SUBAPPLICATION Uebung_HystereseHorizontal_AX_withAnalog (* MID/DEAD/HYSTERESIS-Eingabefelder bewegen live die 5 Schwellwert-Dreiecke im horizontalen Bargraph (wie Uebung_225_AX fuer Workspace_Dreieck, aber 5 Marker statt 1 und mit AR-Arithmetik fuer die 4 abgeleiteten Schwellen) *)
  (* Standard: 61499-2; Description: Copyright (c) 2026 Meisterschulen am Ostbahnhof This program and the accompanying materials are made available under the terms of the Eclipse Public License 2.0 which is available at https://www.eclipse.org/legal/epl-2.0/ SPDX-License-Identifier: EPL-2.0 *)
  (* Version 1.0, 2026-09-26, Franz Höpfinger, Meisterschulen am Ostbahnhof, Franz: 3 Eingabefelder MID/DEAD/HYSTERESIS bewegen die 5 Schwellwert-Dreiecke live - Vorbild Uebung_225_AX (Dreieck-Sollwertmarker): NumericValue_PHYSA -> AR-Arithmetik -> AR_TO_AI -> Q_ChildPosition_AI. *)
  PACKAGE Uebungen;
  IMPORT Uebungen::const::UT::HystereseHorizontal::DefaultPool_Numeric::InputNumber_MID_N;
  IMPORT Uebungen::const::UT::HystereseHorizontal::DefaultPool_Numeric::InputNumber_DEAD_N;
  IMPORT Uebungen::const::UT::HystereseHorizontal::DefaultPool_Numeric::InputNumber_HYSTERESIS_N;
  IMPORT Uebungen::const::UT::HystereseHorizontal::DefaultPool::Polygon_MID;
  IMPORT Uebungen::const::UT::HystereseHorizontal::DefaultPool::Polygon_MID_PLUS_DEAD;
  IMPORT Uebungen::const::UT::HystereseHorizontal::DefaultPool::Polygon_MID_MINUS_DEAD;
  IMPORT Uebungen::const::UT::HystereseHorizontal::DefaultPool::Polygon_MID_PLUS_DEAD_HYST;
  IMPORT Uebungen::const::UT::HystereseHorizontal::DefaultPool::Polygon_MID_MINUS_DEAD_HYST;
  IMPORT Uebungen::const::UT::HystereseHorizontal::DefaultPool::Container_Schwellwerte;
  IMPORT Uebungen::const::UT::HystereseHorizontal::DefaultPool::NumberVariable_Istwert;
  IMPORT logiBUS::io::AI::logiBUS_AI::AnalogInput_I4;
  IMPORT logiBUS::io::DQ::logiBUS_DO::Output_Q1;
  IMPORT logiBUS::io::DQ::logiBUS_DO::Output_Q2;
  FBS
    MID_N : isobus::UT::io::NumericValue::NumericValue_PHYSA(QI := TRUE, stObj := InputNumber_MID_N);
    DEAD_N : isobus::UT::io::NumericValue::NumericValue_PHYSA(QI := TRUE, stObj := InputNumber_DEAD_N);
    HYST_N : isobus::UT::io::NumericValue::NumericValue_PHYSA(QI := TRUE, stObj := InputNumber_HYSTERESIS_N);
    Split_MID : adapter::events::unidirectional::AR_SPLIT_4;
    Split_DEAD : adapter::events::unidirectional::AR_SPLIT_3;
    Split_HYST : adapter::events::unidirectional::AR_SPLIT_3;
    Add_MidDead : adapter::iec61131::arithmetic::AR_ADD_2;
    Sub_MidDead : adapter::iec61131::arithmetic::AR_SUB_2;
    Split_AddResult : adapter::events::unidirectional::AR_SPLIT_2;
    Split_SubResult : adapter::events::unidirectional::AR_SPLIT_2;
    Add_MidDeadHyst : adapter::iec61131::arithmetic::AR_ADD_2;
    Sub_MidDeadHyst : adapter::iec61131::arithmetic::AR_SUB_2;
    AnalogInput_I4 : logiBUS::io::AI::logiBUS_AI_IDA(QI := TRUE, Input := AnalogInput_I4, AnalogInput_hysteresis := DWORD#0, TimeDelta := DWORD#250, TimeRateLimit := DWORD#100);
    AD_TO_AUDI : adapter::conversion::unidirectional::AD_TO_AUDI;
    AUDI_TO_AR : adapter::conversion::unidirectional::AUDI_TO_AR;
    ScaleADC_0_100 : adapter::types::unidirectional::AR::initval::initval_AR(INIT_VAL := REAL#0.024420024420024420);
    Mul_Istwert : adapter::iec61131::arithmetic::AR_MUL_2;
    Split_Istwert : adapter::events::unidirectional::AR_SPLIT_2;
    Q_Istwert : isobus::UT::Q::Q_NumericValue_PHYSA(stObj := (u16ObjId := NumberVariable_Istwert, r32Scale := 1.0, i32Offset := 0, u8Decimals := 0));
    DualHysteresis : logiBUS::signalprocessing::hysteresis::DualHysteresis_AR_AX(QI := TRUE);
    Output_Hoch : logiBUS::io::DQ::logiBUS_QXA(QI := TRUE, Output := Output_Q1);
    Output_Runter : logiBUS::io::DQ::logiBUS_QXA(QI := TRUE, Output := Output_Q2);
    ScalePx_MID : adapter::types::unidirectional::AR::initval::initval_AR(INIT_VAL := REAL#1.86);
    Mul_MID : adapter::iec61131::arithmetic::AR_MUL_2;
    ToAI_MID : adapter::conversion::unidirectional::AR_TO_AI;
    Zero_MID : adapter::types::unidirectional::AI::initval::initval_AI(INIT_VAL := 0);
    QPos_MID : isobus::UT::Q::Q_ChildPosition_AI(u16ObjId := Polygon_MID, u16ObjIdParent := Container_Schwellwerte, xScale := TRUE);
    ScalePx_MID_PLUS_DEAD : adapter::types::unidirectional::AR::initval::initval_AR(INIT_VAL := REAL#1.86);
    Mul_MID_PLUS_DEAD : adapter::iec61131::arithmetic::AR_MUL_2;
    ToAI_MID_PLUS_DEAD : adapter::conversion::unidirectional::AR_TO_AI;
    Zero_MID_PLUS_DEAD : adapter::types::unidirectional::AI::initval::initval_AI(INIT_VAL := 0);
    QPos_MID_PLUS_DEAD : isobus::UT::Q::Q_ChildPosition_AI(u16ObjId := Polygon_MID_PLUS_DEAD, u16ObjIdParent := Container_Schwellwerte, xScale := TRUE);
    ScalePx_MID_MINUS_DEAD : adapter::types::unidirectional::AR::initval::initval_AR(INIT_VAL := REAL#1.86);
    Mul_MID_MINUS_DEAD : adapter::iec61131::arithmetic::AR_MUL_2;
    ToAI_MID_MINUS_DEAD : adapter::conversion::unidirectional::AR_TO_AI;
    Zero_MID_MINUS_DEAD : adapter::types::unidirectional::AI::initval::initval_AI(INIT_VAL := 0);
    QPos_MID_MINUS_DEAD : isobus::UT::Q::Q_ChildPosition_AI(u16ObjId := Polygon_MID_MINUS_DEAD, u16ObjIdParent := Container_Schwellwerte, xScale := TRUE);
    ScalePx_MID_PLUS_DEAD_HYST : adapter::types::unidirectional::AR::initval::initval_AR(INIT_VAL := REAL#1.86);
    Mul_MID_PLUS_DEAD_HYST : adapter::iec61131::arithmetic::AR_MUL_2;
    ToAI_MID_PLUS_DEAD_HYST : adapter::conversion::unidirectional::AR_TO_AI;
    Zero_MID_PLUS_DEAD_HYST : adapter::types::unidirectional::AI::initval::initval_AI(INIT_VAL := 0);
    QPos_MID_PLUS_DEAD_HYST : isobus::UT::Q::Q_ChildPosition_AI(u16ObjId := Polygon_MID_PLUS_DEAD_HYST, u16ObjIdParent := Container_Schwellwerte, xScale := TRUE);
    ScalePx_MID_MINUS_DEAD_HYST : adapter::types::unidirectional::AR::initval::initval_AR(INIT_VAL := REAL#1.86);
    Mul_MID_MINUS_DEAD_HYST : adapter::iec61131::arithmetic::AR_MUL_2;
    ToAI_MID_MINUS_DEAD_HYST : adapter::conversion::unidirectional::AR_TO_AI;
    Zero_MID_MINUS_DEAD_HYST : adapter::types::unidirectional::AI::initval::initval_AI(INIT_VAL := 0);
    QPos_MID_MINUS_DEAD_HYST : isobus::UT::Q::Q_ChildPosition_AI(u16ObjId := Polygon_MID_MINUS_DEAD_HYST, u16ObjIdParent := Container_Schwellwerte, xScale := TRUE);
  END_FBS
  ADAPTER_CONNECTIONS
    MID_N.rPhys TO Split_MID.IN;
    DEAD_N.rPhys TO Split_DEAD.IN;
    HYST_N.rPhys TO Split_HYST.IN;
    Split_MID.OUT2 TO Add_MidDead.IN1;
    Split_DEAD.OUT1 TO Add_MidDead.IN2;
    Split_MID.OUT3 TO Sub_MidDead.IN1;
    Split_DEAD.OUT2 TO Sub_MidDead.IN2;
    Add_MidDead.OUT TO Split_AddResult.IN;
    Sub_MidDead.OUT TO Split_SubResult.IN;
    Split_AddResult.OUT2 TO Add_MidDeadHyst.IN1;
    Split_HYST.OUT1 TO Add_MidDeadHyst.IN2;
    Split_SubResult.OUT2 TO Sub_MidDeadHyst.IN1;
    Split_HYST.OUT2 TO Sub_MidDeadHyst.IN2;
    AnalogInput_I4.IN TO AD_TO_AUDI.AD_IN;
    AD_TO_AUDI.AUDI_OUT TO AUDI_TO_AR.AUDI_IN;
    AUDI_TO_AR.AR_OUT TO Mul_Istwert.IN1;
    ScaleADC_0_100.OUT TO Mul_Istwert.IN2;
    Mul_Istwert.OUT TO Split_Istwert.IN;
    Split_Istwert.OUT1 TO Q_Istwert.rPhys;
    Split_Istwert.OUT2 TO DualHysteresis.INPUT;
    Split_MID.OUT4 TO DualHysteresis.MI;
    Split_DEAD.OUT3 TO DualHysteresis.DEAD;
    Split_HYST.OUT3 TO DualHysteresis.HYSTERESIS;
    DualHysteresis.DO_UP TO Output_Hoch.OUT;
    DualHysteresis.DO_DOWN TO Output_Runter.OUT;
    Split_MID.OUT1 TO Mul_MID.IN1;
    ScalePx_MID.OUT TO Mul_MID.IN2;
    Mul_MID.OUT TO ToAI_MID.AR_IN;
    ToAI_MID.AI_OUT TO QPos_MID.s16Xposition;
    Zero_MID.OUT TO QPos_MID.s16Yposition;
    Split_AddResult.OUT1 TO Mul_MID_PLUS_DEAD.IN1;
    ScalePx_MID_PLUS_DEAD.OUT TO Mul_MID_PLUS_DEAD.IN2;
    Mul_MID_PLUS_DEAD.OUT TO ToAI_MID_PLUS_DEAD.AR_IN;
    ToAI_MID_PLUS_DEAD.AI_OUT TO QPos_MID_PLUS_DEAD.s16Xposition;
    Zero_MID_PLUS_DEAD.OUT TO QPos_MID_PLUS_DEAD.s16Yposition;
    Split_SubResult.OUT1 TO Mul_MID_MINUS_DEAD.IN1;
    ScalePx_MID_MINUS_DEAD.OUT TO Mul_MID_MINUS_DEAD.IN2;
    Mul_MID_MINUS_DEAD.OUT TO ToAI_MID_MINUS_DEAD.AR_IN;
    ToAI_MID_MINUS_DEAD.AI_OUT TO QPos_MID_MINUS_DEAD.s16Xposition;
    Zero_MID_MINUS_DEAD.OUT TO QPos_MID_MINUS_DEAD.s16Yposition;
    Add_MidDeadHyst.OUT TO Mul_MID_PLUS_DEAD_HYST.IN1;
    ScalePx_MID_PLUS_DEAD_HYST.OUT TO Mul_MID_PLUS_DEAD_HYST.IN2;
    Mul_MID_PLUS_DEAD_HYST.OUT TO ToAI_MID_PLUS_DEAD_HYST.AR_IN;
    ToAI_MID_PLUS_DEAD_HYST.AI_OUT TO QPos_MID_PLUS_DEAD_HYST.s16Xposition;
    Zero_MID_PLUS_DEAD_HYST.OUT TO QPos_MID_PLUS_DEAD_HYST.s16Yposition;
    Sub_MidDeadHyst.OUT TO Mul_MID_MINUS_DEAD_HYST.IN1;
    ScalePx_MID_MINUS_DEAD_HYST.OUT TO Mul_MID_MINUS_DEAD_HYST.IN2;
    Mul_MID_MINUS_DEAD_HYST.OUT TO ToAI_MID_MINUS_DEAD_HYST.AR_IN;
    ToAI_MID_MINUS_DEAD_HYST.AI_OUT TO QPos_MID_MINUS_DEAD_HYST.s16Xposition;
    Zero_MID_MINUS_DEAD_HYST.OUT TO QPos_MID_MINUS_DEAD_HYST.s16Yposition;
  END_CONNECTIONS
END_SUBAPPLICATION
